FUNCTION_BLOCK FB_PositionX IMPLEMENTS IPosition
VAR_INPUT
END_VAR
VAR_OUTPUT
END_VAR
VAR
	_position	: LREAL;
	_linked		: UDINT;
END_VAR

METHOD Available : BOOL
IF _linked = 0 THEN
	Available := TRUE;
END_IF
END_METHOD

METHOD SetMover : BOOL
VAR_INPUT
	moverNumber	: UDINT;
END_VAR
IF _linked = 0 AND moverNumber <> 0 THEN
	_linked := moverNumber;
	SetMover := TRUE;
END_IF
END_METHOD

METHOD SetPosition
VAR_INPUT
	position	: LREAL;
END_VAR
_position := position;
END_METHOD

END_FUNCTION_BLOCK

(* stored: Version 1.1.0.1, ProductVersion 3.1.4026.12
   POU FB_PositionX: Id {f9da956f-0a89-4671-827d-6c04f2d33aac}, SpecialFunc None
   Method Available: Id {8b398280-858b-4913-9249-673e7096f588}
   Method SetMover: Id {83289a63-eb24-4eac-83c4-eebaa2247582}
   Method SetPosition: Id {66d03994-61db-4326-a0b5-789123102fd6} *)
